Omron CX-Programmer project NewProject (CX-Programmer 9.75)

# PLC NewPLC1: CP2E-N N

## Global symbols (name address type ; comment)
W1.01 BOOL  ; MieKering_Picked
FB_MODBUSTCP_SERVER _CP2E003_ExecuteModTcpServer

## Program NewProgram1 (cyclic task 0)

### Section Section1

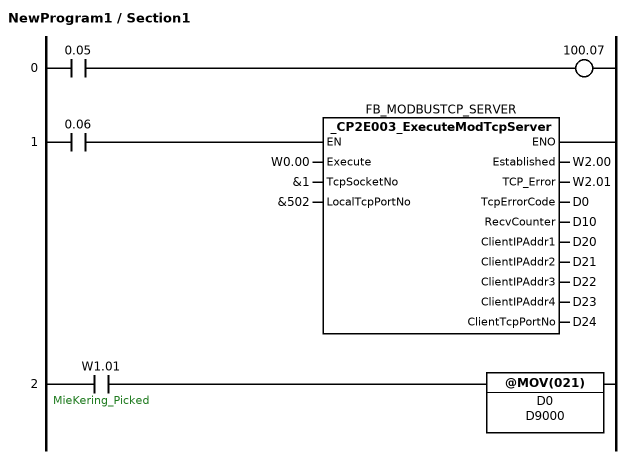
; rung 0
LD 0.05
OUT 100.07
; rung 1
LD 0.06
CALL FB_MODBUSTCP_SERVER : _CP2E003_ExecuteModTcpServer (Execute := W0.00, TcpSocketNo := &1, LocalTcpPortNo := &502, Established => W2.00, TCP_Error => W2.01, TcpErrorCode => D0, RecvCounter => D10, ClientIPAddr1 => D20, ClientIPAddr2 => D21, ClientIPAddr3 => D22, ClientIPAddr4 => D23, ClientTcpPortNo => D24)
; rung 2
LD W1.01  ; MieKering_Picked
@MOV(021) D0 D9000

### Section END
; rung 0
END(001)

## Function block _CP2E003_ExecuteModTcpServer (Omron library block, body left out)